(* IEC 61131-3 sources: POLSL-Mgr-ST-Compiler/benchmark/delay, 1 file *)

(* ---- delay.st ---- *)
PROGRAM main
    VAR
        counter: LINT;
    END_VAR

    counter := LINT#100_000;

    WHILE counter >= LINT#0 DO
        counter := counter - LINT#1;
    END_WHILE;
END_PROGRAM
